// TIA Portal V19 export
TYPE "LAF_typeAxisDiagStatus"
TITLE = LAF_typeAxisDiagStatus
// Status information, warnings and errors of a Technology Object
// stored: Access Published
   STRUCT
      statusWord { ExternalWritable := 'False'} : DWord;   // Status word of the technology object
      statusWord2 { ExternalWritable := 'False'} : DWord;   // Status word 2 of the technology object
      warningWord { ExternalWritable := 'False'} : DWord;   // Warning word of the technology object
      errorWord { ExternalWritable := 'False'} : DWord;   // Error word of the technology object
      status { ExternalWritable := 'False'} : "LAF_typeAxisDiagStatusWord";
      status2 { ExternalWritable := 'False'} : "LAF_typeAxisDiagStatusWord2";
      warning { ExternalWritable := 'False'} : "LAF_typeAxisDiagWarningWord";
      error { ExternalWritable := 'False'} : "LAF_typeAxisDiagErrorWord";
      errorDetail { ExternalWritable := 'False'} : "LAF_typeAxisDiagErrorDetail";
   END_STRUCT;
END_TYPE
